INTERFACE I_MotionDrive

PROPERTY Busy : BOOL
GET
END_GET
SET
END_SET
END_PROPERTY

PROPERTY CustomErrorMessage : T_MAXSTRING
GET
END_GET
SET
END_SET
END_PROPERTY

METHOD DepsInit
VAR_INPUT
END_VAR
END_METHOD

PROPERTY Done : BOOL
GET
END_GET
SET
END_SET
END_PROPERTY

METHOD EncRestore
VAR_INPUT
END_VAR
END_METHOD

METHOD EncSave
VAR_INPUT
END_VAR
END_METHOD

PROPERTY Error : BOOL
GET
END_GET
SET
END_SET
END_PROPERTY

PROPERTY ErrorCode : UDINT
GET
END_GET
SET
END_SET
END_PROPERTY

METHOD GetInterlocksRef
VAR_INPUT
END_VAR
END_METHOD


METHOD GetLoggerRef : REFERENCE TO AXIS_REF
END_METHOD

METHOD GetPersistantStorageRef
VAR_INPUT
END_VAR
END_METHOD

METHOD HomeCmd
VAR_INPUT
END_VAR
END_METHOD


METHOD MoveAbsolute
VAR_INPUT
    Position : LREAL; 
    Velocity : LREAL; 
    Acceleration : LREAL := 0.0; 
    Deceleration : LREAL := 0.0; 
    Jerk : LREAL := 0.0;
    BufferMode : MC_BufferMode := MC_BufferMode.MC_Aborting;
END_VAR
VAR_OUTPUT
    Done : BOOL;
    Busy : BOOL;
    Active : BOOL;
    CommandAborted : BOOL;
    Error : BOOL;
    ErrorID : UDINT;
    ErrorStr : T_MaxString;
END_VAR
END_METHOD

METHOD MoveCmd
VAR_INPUT
END_VAR
END_METHOD

PROPERTY Name : STRING
GET
END_GET
SET
END_SET
END_PROPERTY

METHOD NCParamsExposed
VAR_INPUT
END_VAR
END_METHOD

METHOD NCStatusExposed
VAR_INPUT
END_VAR
END_METHOD

PROPERTY NegGoal : BOOL
GET
END_GET
SET
END_SET
END_PROPERTY

PROPERTY PosGoal : BOOL
GET
END_GET
SET
END_SET
END_PROPERTY

METHOD PostMoveHandling
VAR_INPUT
END_VAR
END_METHOD

METHOD ProcessMoveReq
VAR_INPUT
END_VAR
END_METHOD

END_INTERFACE

(* stored: Version 1.1.0.1
   Itf I_MotionDrive: Id {4f84f724-7938-4847-ac53-18866323f75e}
   Property Busy: Id {d927182d-eff1-4072-9dbb-b154fb0b0384}
   Get Get: Id {5caf1a60-abb0-4745-b78d-031d87326f3a}
   Set Set: Id {6babf4a2-d1a1-4509-8880-abc134803329}
   Property CustomErrorMessage: Id {1f202727-1b36-4e25-b74c-103d33b9d571}
   Get Get: Id {f8e06972-f73d-4bc3-9676-e2259d72e3ee}
   Set Set: Id {aae53a41-e997-4a33-a47e-083bd72a85ca}
   Method DepsInit: Id {bf5827d1-d917-4cf2-bee1-86b0b5256fcf}
   Property Done: Id {3f8a8de7-7e6f-415e-90b3-ae5922bd3074}
   Get Get: Id {e0481405-1904-426f-8294-683a0a15ba2c}
   Set Set: Id {69ec95aa-0883-4c80-92a1-83f7f5d53e54}
   Method EncRestore: Id {2381ad33-db9f-4502-8f18-42d9f37ce4d4}
   Method EncSave: Id {10587d60-0d31-4f6e-bd02-f4dc5980cb00}
   Property Error: Id {28692bda-2e15-49a9-ae9c-44ee2c225402}
   Get Get: Id {e7c06eb5-1986-4004-bdcb-ca18cd302e3f}
   Set Set: Id {5320cbe2-83f6-49ab-a814-bb332a3d0b75}
   Property ErrorCode: Id {415dcb0a-1a80-4f20-a5f6-d07b913efdcb}
   Get Get: Id {2080dd72-b57e-4aae-b589-16fc55f2d7f8}
   Set Set: Id {eb8abf2e-d9e9-4d6c-a6ee-9a201b51f0c5}
   Method GetInterlocksRef: Id {3cfdd636-3485-4b90-82df-1f6314019050}
   Method GetLoggerRef: Id {f7a7f054-d0c4-4c97-8fd2-100c34cb6c54}
   Method GetPersistantStorageRef: Id {7e64d835-954c-4a5e-989c-ebb2ac7815a4}
   Method HomeCmd: Id {9fdc0c70-7fd4-4e1d-973a-5fd32a2ffa74}
   Method MoveAbsolute: Id {1eeced1d-efd0-4ca8-90ed-573a0f3007ea}
   Method MoveCmd: Id {34c1c090-b9ee-44c1-a1e3-f9de462d94e8}
   Property Name: Id {808bc845-b6e4-4963-ab8f-244d15a3cc40}
   Get Get: Id {eef700d5-67cb-4093-abd3-49b2850feb0c}
   Set Set: Id {a8ad97b6-7dbe-4ad8-a2ac-9e24c41ccebb}
   Method NCParamsExposed: Id {abf9dd67-1532-4b48-ba74-a21084aac3ca}
   Method NCStatusExposed: Id {0fbeb893-2508-4c58-8356-be243474fc34}
   Property NegGoal: Id {8ca9aaff-70e5-4a7d-a380-f334afbad2d7}
   Get Get: Id {dcb0f332-0cee-463b-a760-dfbb09a2481f}
   Set Set: Id {b6d4edb5-1521-4c30-ad4f-617130ebe079}
   Property PosGoal: Id {3bbc2f55-6d26-4fcf-84a1-58d794d496f9}
   Get Get: Id {c16d3cd5-bc57-4e01-b657-b628634e13d4}
   Set Set: Id {ab4cb165-b4bb-475f-901a-3072d677c7cc}
   Method PostMoveHandling: Id {da3cb092-448a-4700-855b-582d56530d50}
   Method ProcessMoveReq: Id {16636825-34ac-44bb-b4de-2566f4d18b17} *)
